// TIA Portal project "S7-LAD-P1-MINI-ENG Bit logic operations 04 Template" (V16)
// Vorlageprojekt für das Buch mit Zielsystem S7-1200

(* hardware
DEVICE "S7-1200-Station_1"  S7-1200 Station
   slot 0: "Baugruppenträger_0"  Rack  V1.0
   slot 1: "PLC_1"  CPU 1211C DC/DC/DC  6ES7 211-1AE40-0XB0  V4.1
*)

// ===== PLC "PLC_1"  CPU 1211C DC/DC/DC =====

VAR_GLOBAL   // PLC tag table "Standard-Variablentabelle"
   "xConveyor_forward" AT %A0.0 : Bool;
   "xPushButton_Start" AT %E0.0 : Bool;
   "xPushButton_stop" AT %E0.1 : Bool;
   "xSensor_1" AT %I0.2 : Bool;
   "xSelector_Enable" AT %I0.3 : Bool;
   "xSensor_2" AT %I0.4 : Bool;
   "xConveyor_Backward" AT %Q0.5 : Bool;
END_VAR

FUNCTION "MHJ-PLC-Lab-Function-S71200" : Void   // FC9000, SCL
{ S7_Optimized_Access := 'TRUE' }
VERSION : 0.1
   VAR_TEMP
      rdTimeReturn : Int;
      outputTime : DTL;
      SyncVal : Byte;
      forVal : Int;
      forVal_2 : Int;
      Value : Byte;
   END_VAR
   VAR CONSTANT
      CompVal : Byte := 16#34;
      Value_01 : Byte := 16#11;
      Value_01_DW : DWord := 16#A165_D992;
      Value_02_DW : DWord := 16#58BE_4401;
   END_VAR
BEGIN

   #Value:=PEEK(area := 16#82,
        dbNumber := 0,
        byteOffset := 511);
   #Value := #Value + 1;

   POKE(area := 16#82,
        dbNumber := 0,
        byteOffset := 511,
        value := #Value);

   POKE(area:=16#81,
        dbNumber:=0,
        byteOffset:=1016,
        value:=#Value_01_DW);
   POKE(area := 16#81,
        dbNumber := 0,
        byteOffset := 1020,
        value := #Value_02_DW);

   POKE(area := 16#81,
        dbNumber := 0,
        byteOffset := 511,
        value := B#16#00);

   FOR #forVal := 0 TO 120 DO
       FOR #forVal_2:=0 TO 10 DO
           #rdTimeReturn:=RD_SYS_T(#outputTime);
           #rdTimeReturn := WR_SYS_T(#outputTime);
           #rdTimeReturn := RD_SYS_T(#outputTime);
           #rdTimeReturn := WR_SYS_T(#outputTime);
       END_FOR;
       #SyncVal:= PEEK(area := 16#81,
                      dbNumber := 0,
                      byteOffset := 511);
       IF #SyncVal = #CompVal THEN
          GOTO M_1;
       END_IF;
   END_FOR;
   RETURN;

   M_1:
   POKE(area := 16#81,
        dbNumber := 0,
        byteOffset := 511,
        value := B#16#0);
END_FUNCTION

ORGANIZATION_BLOCK "Main"   // OB1, LAD, ProgramCycle
TITLE = "Main Program Sweep (Cycle)"
{ S7_Optimized_Access := 'TRUE' }
VERSION : 0.1
   VAR_INPUT
      Initial_Call : Bool;   // Initial call of this OB
      Remanence : Bool;   // =True, if remanent data are available
   END_VAR
BEGIN

REGION Network 1
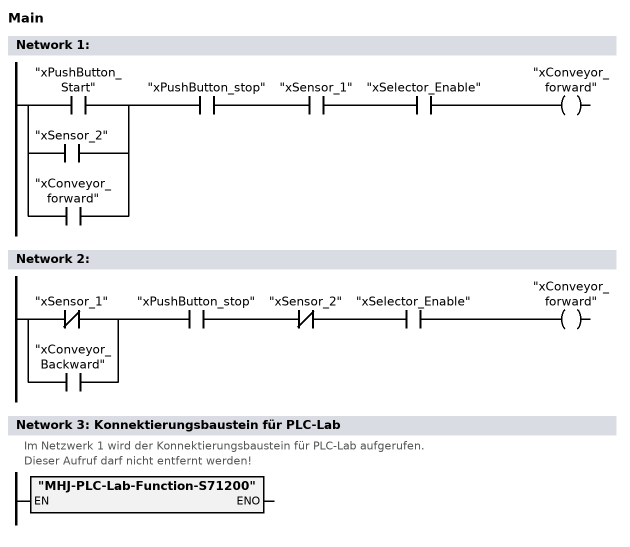
   RUNG wire#powerrail
      Contact( "xPushButton_Start" )
      wire#w1
      Contact( "xPushButton_stop" )
      Contact( "xSensor_1" )
      Contact( "xSelector_Enable" )
      Coil( "xConveyor_forward" )
   END_RUNG
   RUNG wire#powerrail
      Contact( "xSensor_2" )
   END_RUNG wire#w1
   RUNG wire#powerrail
      Contact( "xConveyor_forward" )
   END_RUNG wire#w1
   // the same network as SCL:
   "xConveyor_forward" := ("xPushButton_Start" OR "xSensor_2" OR "xConveyor_forward") AND "xPushButton_stop" AND "xSensor_1" AND "xSelector_Enable";
END_REGION

REGION Network 2
   RUNG wire#powerrail
      I_Contact( "xSensor_1" )
      wire#w1
      Contact( "xPushButton_stop" )
      I_Contact( "xSensor_2" )
      Contact( "xSelector_Enable" )
      Coil( "xConveyor_forward" )
   END_RUNG
   RUNG wire#powerrail
      Contact( "xConveyor_Backward" )
   END_RUNG wire#w1
   // the same network as SCL:
   "xConveyor_forward" := (NOT "xSensor_1" OR "xConveyor_Backward") AND "xPushButton_stop" AND NOT "xSensor_2" AND "xSelector_Enable";
END_REGION

REGION Network 3: Konnektierungsbaustein für PLC-Lab
   // Im Netzwerk 1 wird der Konnektierungsbaustein für PLC-Lab aufgerufen.
   // Dieser Aufruf darf nicht entfernt werden!
   RUNG wire#powerrail
      "MHJ-PLC-Lab-Function-S71200"()
   END_RUNG
   // the same network as SCL:
   "MHJ-PLC-Lab-Function-S71200"();
END_REGION
END_ORGANIZATION_BLOCK